(* IEC 61131-3 sources: volt/packages/volt-lsp-iec/test-corpus/pro2193/Device/Plc Logic/Application/03 Hardware Units/32 BFU/32.70 - Box Pusher, 1 file *)

(* ---- BoxPushers.pou ---- *)
{attribute 'symbol' := 'none'}
PROGRAM BoxPushers
VAR_INPUT
	{attribute 'symbol' := 'readwrite'}	Unit						: ARRAY[1..usiNumberOfUnits] OF BoxPusher_DefaultFB
	[
		(
			instanceNo		:= 1,
			moduleManager	:= GlobalVars_BFU.fbModuleManager,
			moduleParent	:= 0,
			resetCondition1	:= 0,
			resetCondition2	:= 0,
		)
	];

END_VAR
VAR
	i							: USINT;
END_VAR
VAR RETAIN PERSISTENT
	{attribute 'symbol' := 'readwrite'}	Data						: ARRAY[1..BoxPushers.usiNumberOfUnits] OF BoxPusher_Default_DataType;
END_VAR
VAR CONSTANT
	usiNumberOfUnits			: USINT := 1;
END_VAR

%LANGUAGE ST
FOR i := 1 TO usiNumberOfUnits DO
	Unit[i](
		Data						:= Data[i],
		BoxInFillPosition			:= BoxCenterUnits.Unit[1].BoxInFillPosition);
END_FOR

END_PROGRAM
